Fanuc KAREL source: kt00991.KL

-- PROVISIONAL review KL for V1013-1; original PC SHA256 e5529cb71040a6be81702ad9ef5f71471304df56c701fc133019c3da4b605255
-- Incomplete behavior may be omitted. Consult companion uncertainty JSON. Do not deploy.
PROGRAM KT00991
%NOLOCKGROUP
VAR
  X : REAL
  Y : REAL
  Z : REAL
  W : REAL
  P : REAL
  R : REAL
-- UNRESOLVED_DECL P1 type=000101
-- UNRESOLVED_DECL P2 type=000101
-- UNRESOLVED_DECL CFG type=00001c
BEGIN
  -- UNRESOLVED_PC offsets 5-65; opcodes 27,27,49,7E,AD,22,22,22,22,22,22,22,76
  -- UNRESOLVED_PC offsets 70-74; opcodes 7F
END KT00991
